// TIA Portal V16 export
// export: Created 2022-03-28T07:44:04.7254911Z, ExportSetting WithDefaults, DisplayName Totally Integrated Automation Portal, DisplayVersion V16 Update 5, DisplayName TIA Portal Version Control Interface, DisplayVersion V16 Update 2, DisplayName TIA Portal Openness, DisplayVersion V16 Update 5, DisplayName STEP 7 Professional, DisplayVersion V16 Update 5, DisplayName STEP 7 Safety, DisplayVersion V16, DisplayName WinCC Professional, DisplayVersion V16 Update 5
FUNCTION "fc_02_Outputs" : Void   // FC2, LAD
{ S7_Optimized_Access := 'TRUE' }
VERSION : 0.1
// stored: AutoNumber false, IsIECCheckEnabled false, SetENOAutomatically false, UDAEnableTagReadback false
   VAR_TEMP
      bIsInverted : Bool;
   END_VAR
   VAR_TEMP   // added for the SCL form of the ladder/FBD networks
      _w1 : Bool;
      _w2 : Bool;
      _w3 : Bool;
      _w4 : Bool;
   END_VAR
BEGIN

REGION Network 1: Rele rearme
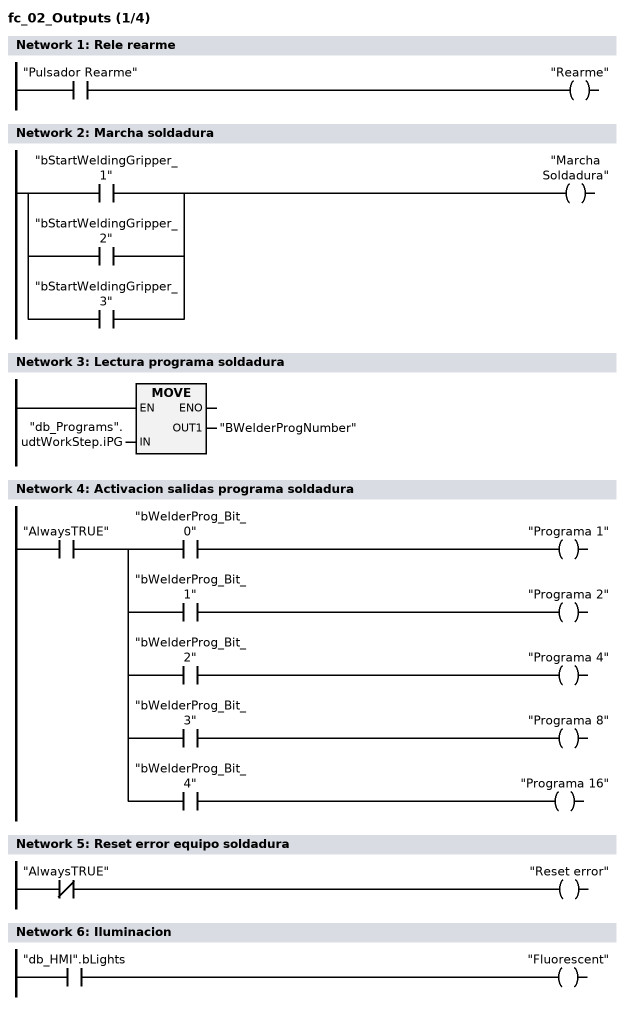
   RUNG wire#powerrail
      Contact( "Pulsador Rearme" )
      Coil( "Rearme" )
   END_RUNG
   // the same network as SCL:
   "Rearme" := "Pulsador Rearme";
END_REGION

REGION Network 2: Marcha soldadura
   RUNG wire#powerrail
      Contact( "bStartWeldingGripper_1" )
      wire#w1
      Coil( "Marcha Soldadura" )
   END_RUNG
   RUNG wire#powerrail
      Contact( "bStartWeldingGripper_2" )
   END_RUNG wire#w1
   RUNG wire#powerrail
      Contact( "bStartWeldingGripper_3" )
   END_RUNG wire#w1
   // the same network as SCL:
   "Marcha Soldadura" := "bStartWeldingGripper_1" OR "bStartWeldingGripper_2" OR "bStartWeldingGripper_3";
END_REGION

REGION Network 3: Lectura programa soldadura
   RUNG wire#powerrail
      Move(in := "db_Programs".udtWorkStep.iPG, out1 => "BWelderProgNumber")
   END_RUNG
   // the same network as SCL:
   "BWelderProgNumber" := "db_Programs".udtWorkStep.iPG;
END_REGION

REGION Network 4: Activacion salidas programa soldadura
   RUNG wire#powerrail
      Contact( "AlwaysTRUE" )
      wire#w1
      Contact( "bWelderProg_Bit_0" )
      Coil( "Programa 1" )
   END_RUNG
   RUNG wire#w1
      Contact( "bWelderProg_Bit_1" )
      Coil( "Programa 2" )
   END_RUNG
   RUNG wire#w1
      Contact( "bWelderProg_Bit_2" )
      Coil( "Programa 4" )
   END_RUNG
   RUNG wire#w1
      Contact( "bWelderProg_Bit_3" )
      Coil( "Programa 8" )
   END_RUNG
   RUNG wire#w1
      Contact( "bWelderProg_Bit_4" )
      Coil( "Programa 16" )
   END_RUNG
   // the same network as SCL:
   "Programa 1" := "AlwaysTRUE" AND "bWelderProg_Bit_0";
   "Programa 2" := "AlwaysTRUE" AND "bWelderProg_Bit_1";
   "Programa 4" := "AlwaysTRUE" AND "bWelderProg_Bit_2";
   "Programa 8" := "AlwaysTRUE" AND "bWelderProg_Bit_3";
   "Programa 16" := "AlwaysTRUE" AND "bWelderProg_Bit_4";
END_REGION

REGION Network 5: Reset error equipo soldadura
   RUNG wire#powerrail
      I_Contact( "AlwaysTRUE" )
      Coil( "Reset error" )
   END_RUNG
   // the same network as SCL:
   "Reset error" := NOT "AlwaysTRUE";
END_REGION

REGION Network 6: Iluminacion
   RUNG wire#powerrail
      Contact( "db_HMI".bLights )
      Coil( "Fluorescent" )
   END_RUNG
   // the same network as SCL:
   "Fluorescent" := "db_HMI".bLights;
END_REGION

REGION Network 7: Pilotos 1
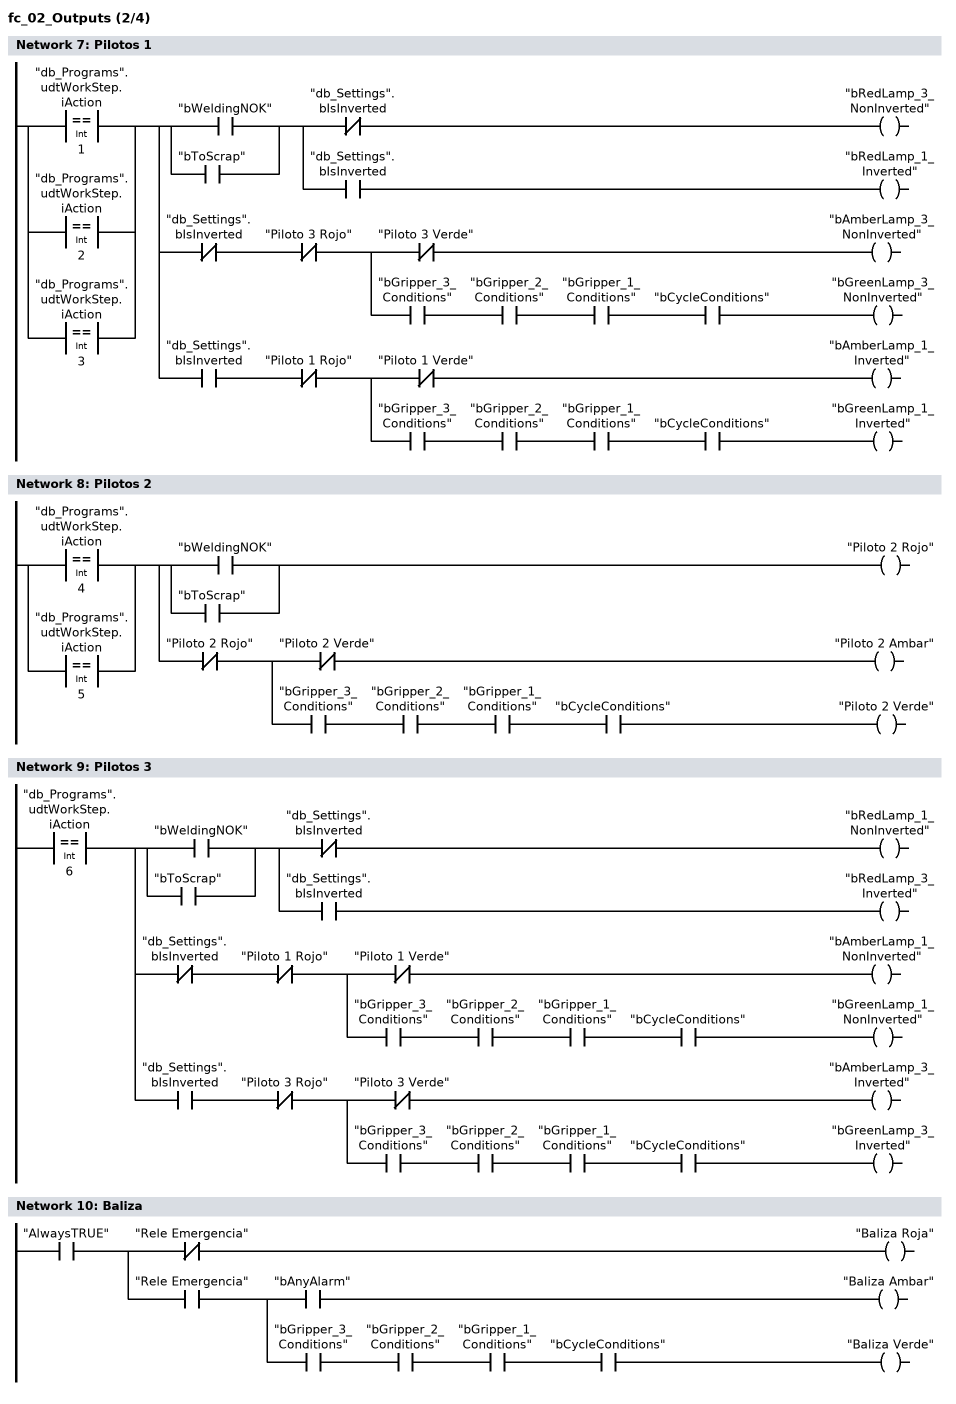
   RUNG wire#powerrail
      { S7_Templates := "SrcType := Int" } EQ_Contact(in1 := "db_Programs".udtWorkStep.iAction, in2 := 1)
      wire#w1
      Contact( "bWeldingNOK" )
      wire#w2
      I_Contact( "db_Settings".bIsInverted )
      Coil( "bRedLamp_3_NonInverted" )
   END_RUNG
   RUNG wire#powerrail
      { S7_Templates := "SrcType := Int" } EQ_Contact(in1 := "db_Programs".udtWorkStep.iAction, in2 := 2)
   END_RUNG wire#w1
   RUNG wire#powerrail
      { S7_Templates := "SrcType := Int" } EQ_Contact(in1 := "db_Programs".udtWorkStep.iAction, in2 := 3)
   END_RUNG wire#w1
   RUNG wire#w1
      Contact( "bToScrap" )
   END_RUNG wire#w2
   RUNG wire#w2
      Contact( "db_Settings".bIsInverted )
      Coil( "bRedLamp_1_Inverted" )
   END_RUNG
   RUNG wire#w1
      I_Contact( "db_Settings".bIsInverted )
      I_Contact( "Piloto 3 Rojo" )
      wire#w3
      I_Contact( "Piloto 3 Verde" )
      Coil( "bAmberLamp_3_NonInverted" )
   END_RUNG
   RUNG wire#w3
      Contact( "bGripper_3_Conditions" )
      Contact( "bGripper_2_Conditions" )
      Contact( "bGripper_1_Conditions" )
      Contact( "bCycleConditions" )
      Coil( "bGreenLamp_3_NonInverted" )
   END_RUNG
   RUNG wire#w1
      Contact( "db_Settings".bIsInverted )
      I_Contact( "Piloto 1 Rojo" )
      wire#w4
      I_Contact( "Piloto 1 Verde" )
      Coil( "bAmberLamp_1_Inverted" )
   END_RUNG
   RUNG wire#w4
      Contact( "bGripper_3_Conditions" )
      Contact( "bGripper_2_Conditions" )
      Contact( "bGripper_1_Conditions" )
      Contact( "bCycleConditions" )
      Coil( "bGreenLamp_1_Inverted" )
   END_RUNG
   // the same network as SCL:
   #_w1 := ("db_Programs".udtWorkStep.iAction = 1) OR ("db_Programs".udtWorkStep.iAction = 2) OR ("db_Programs".udtWorkStep.iAction = 3);
   #_w2 := #_w1 AND ("bWeldingNOK" OR "bToScrap");
   "bRedLamp_3_NonInverted" := #_w2 AND NOT "db_Settings".bIsInverted;
   "bRedLamp_1_Inverted" := #_w2 AND "db_Settings".bIsInverted;
   #_w3 := #_w1 AND NOT "db_Settings".bIsInverted AND NOT "Piloto 3 Rojo";
   "bAmberLamp_3_NonInverted" := #_w3 AND NOT "Piloto 3 Verde";
   "bGreenLamp_3_NonInverted" := #_w3 AND "bGripper_3_Conditions" AND "bGripper_2_Conditions" AND "bGripper_1_Conditions" AND "bCycleConditions";
   #_w4 := #_w1 AND "db_Settings".bIsInverted AND NOT "Piloto 1 Rojo";
   "bAmberLamp_1_Inverted" := #_w4 AND NOT "Piloto 1 Verde";
   "bGreenLamp_1_Inverted" := #_w4 AND "bGripper_3_Conditions" AND "bGripper_2_Conditions" AND "bGripper_1_Conditions" AND "bCycleConditions";
END_REGION

REGION Network 8: Pilotos 2
   RUNG wire#powerrail
      { S7_Templates := "SrcType := Int" } EQ_Contact(in1 := "db_Programs".udtWorkStep.iAction, in2 := 4)
      wire#w1
      Contact( "bWeldingNOK" )
      wire#w2
      Coil( "Piloto 2 Rojo" )
   END_RUNG
   RUNG wire#powerrail
      { S7_Templates := "SrcType := Int" } EQ_Contact(in1 := "db_Programs".udtWorkStep.iAction, in2 := 5)
   END_RUNG wire#w1
   RUNG wire#w1
      Contact( "bToScrap" )
   END_RUNG wire#w2
   RUNG wire#w1
      I_Contact( "Piloto 2 Rojo" )
      wire#w3
      I_Contact( "Piloto 2 Verde" )
      Coil( "Piloto 2 Ambar" )
   END_RUNG
   RUNG wire#w3
      Contact( "bGripper_3_Conditions" )
      Contact( "bGripper_2_Conditions" )
      Contact( "bGripper_1_Conditions" )
      Contact( "bCycleConditions" )
      Coil( "Piloto 2 Verde" )
   END_RUNG
   // the same network as SCL:
   #_w1 := ("db_Programs".udtWorkStep.iAction = 4) OR ("db_Programs".udtWorkStep.iAction = 5);
   "Piloto 2 Rojo" := #_w1 AND ("bWeldingNOK" OR "bToScrap");
   #_w2 := #_w1 AND NOT "Piloto 2 Rojo";
   "Piloto 2 Ambar" := #_w2 AND NOT "Piloto 2 Verde";
   "Piloto 2 Verde" := #_w2 AND "bGripper_3_Conditions" AND "bGripper_2_Conditions" AND "bGripper_1_Conditions" AND "bCycleConditions";
END_REGION

REGION Network 9: Pilotos 3
   RUNG wire#powerrail
      { S7_Templates := "SrcType := Int" } EQ_Contact(in1 := "db_Programs".udtWorkStep.iAction, in2 := 6)
      wire#w1
      Contact( "bWeldingNOK" )
      wire#w2
      I_Contact( "db_Settings".bIsInverted )
      Coil( "bRedLamp_1_NonInverted" )
   END_RUNG
   RUNG wire#w1
      Contact( "bToScrap" )
   END_RUNG wire#w2
   RUNG wire#w2
      Contact( "db_Settings".bIsInverted )
      Coil( "bRedLamp_3_Inverted" )
   END_RUNG
   RUNG wire#w1
      I_Contact( "db_Settings".bIsInverted )
      I_Contact( "Piloto 1 Rojo" )
      wire#w3
      I_Contact( "Piloto 1 Verde" )
      Coil( "bAmberLamp_1_NonInverted" )
   END_RUNG
   RUNG wire#w3
      Contact( "bGripper_3_Conditions" )
      Contact( "bGripper_2_Conditions" )
      Contact( "bGripper_1_Conditions" )
      Contact( "bCycleConditions" )
      Coil( "bGreenLamp_1_NonInverted" )
   END_RUNG
   RUNG wire#w1
      Contact( "db_Settings".bIsInverted )
      I_Contact( "Piloto 3 Rojo" )
      wire#w4
      I_Contact( "Piloto 3 Verde" )
      Coil( "bAmberLamp_3_Inverted" )
   END_RUNG
   RUNG wire#w4
      Contact( "bGripper_3_Conditions" )
      Contact( "bGripper_2_Conditions" )
      Contact( "bGripper_1_Conditions" )
      Contact( "bCycleConditions" )
      Coil( "bGreenLamp_3_Inverted" )
   END_RUNG
   // the same network as SCL:
   #_w1 := "db_Programs".udtWorkStep.iAction = 6;
   #_w2 := #_w1 AND ("bWeldingNOK" OR "bToScrap");
   "bRedLamp_1_NonInverted" := #_w2 AND NOT "db_Settings".bIsInverted;
   "bRedLamp_3_Inverted" := #_w2 AND "db_Settings".bIsInverted;
   #_w3 := #_w1 AND NOT "db_Settings".bIsInverted AND NOT "Piloto 1 Rojo";
   "bAmberLamp_1_NonInverted" := #_w3 AND NOT "Piloto 1 Verde";
   "bGreenLamp_1_NonInverted" := #_w3 AND "bGripper_3_Conditions" AND "bGripper_2_Conditions" AND "bGripper_1_Conditions" AND "bCycleConditions";
   #_w4 := #_w1 AND "db_Settings".bIsInverted AND NOT "Piloto 3 Rojo";
   "bAmberLamp_3_Inverted" := #_w4 AND NOT "Piloto 3 Verde";
   "bGreenLamp_3_Inverted" := #_w4 AND "bGripper_3_Conditions" AND "bGripper_2_Conditions" AND "bGripper_1_Conditions" AND "bCycleConditions";
END_REGION

REGION Network 10: Baliza
   RUNG wire#powerrail
      Contact( "AlwaysTRUE" )
      wire#w1
      I_Contact( "Rele Emergencia" )
      Coil( "Baliza Roja" )
   END_RUNG
   RUNG wire#w1
      Contact( "Rele Emergencia" )
      wire#w2
      Contact( "bAnyAlarm" )
      Coil( "Baliza Ambar" )
   END_RUNG
   RUNG wire#w2
      Contact( "bGripper_3_Conditions" )
      Contact( "bGripper_2_Conditions" )
      Contact( "bGripper_1_Conditions" )
      Contact( "bCycleConditions" )
      Coil( "Baliza Verde" )
   END_RUNG
   // the same network as SCL:
   "Baliza Roja" := "AlwaysTRUE" AND NOT "Rele Emergencia";
   #_w1 := "AlwaysTRUE" AND "Rele Emergencia";
   "Baliza Ambar" := #_w1 AND "bAnyAlarm";
   "Baliza Verde" := #_w1 AND "bGripper_3_Conditions" AND "bGripper_2_Conditions" AND "bGripper_1_Conditions" AND "bCycleConditions";
END_REGION

REGION Network 11: Piloto rearme
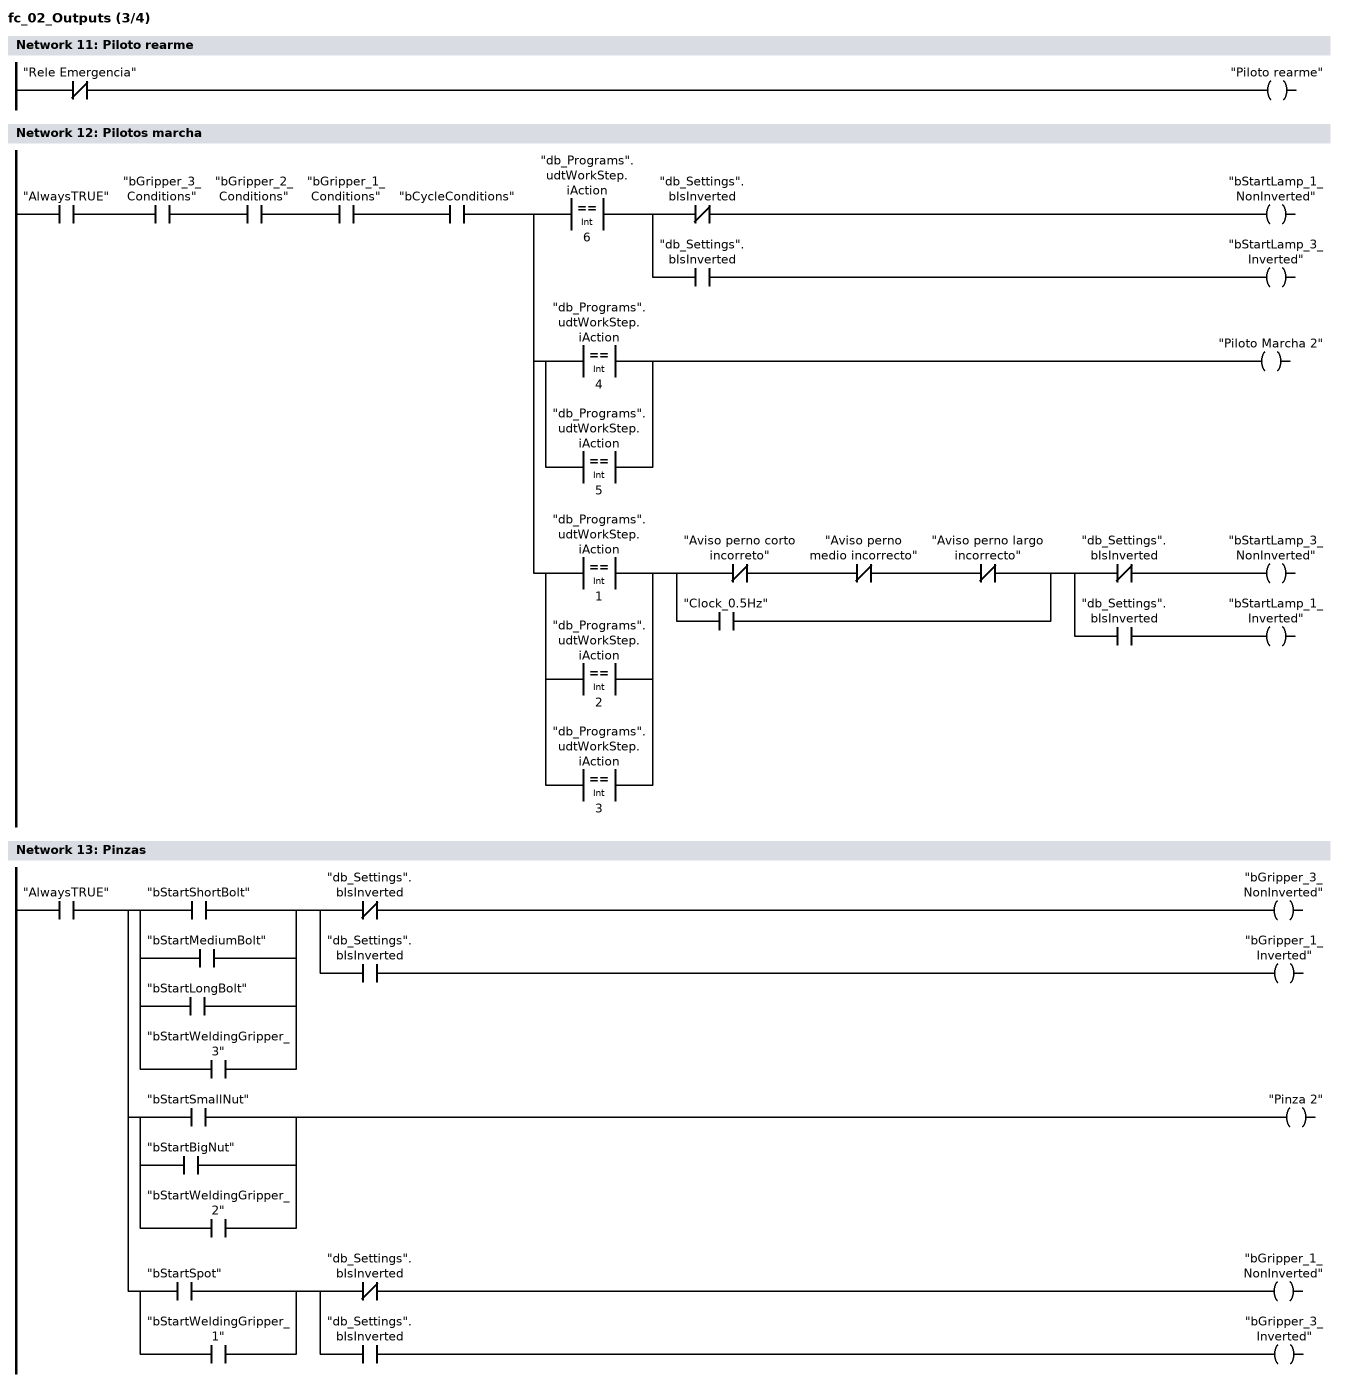
   RUNG wire#powerrail
      I_Contact( "Rele Emergencia" )
      Coil( "Piloto rearme" )
   END_RUNG
   // the same network as SCL:
   "Piloto rearme" := NOT "Rele Emergencia";
END_REGION

REGION Network 12: Pilotos marcha
   RUNG wire#powerrail
      Contact( "AlwaysTRUE" )
      Contact( "bGripper_3_Conditions" )
      Contact( "bGripper_2_Conditions" )
      Contact( "bGripper_1_Conditions" )
      Contact( "bCycleConditions" )
      wire#w1
      { S7_Templates := "SrcType := Int" } EQ_Contact(in1 := "db_Programs".udtWorkStep.iAction, in2 := 6)
      wire#w2
      I_Contact( "db_Settings".bIsInverted )
      Coil( "bStartLamp_1_NonInverted" )
   END_RUNG
   RUNG wire#w2
      Contact( "db_Settings".bIsInverted )
      Coil( "bStartLamp_3_Inverted" )
   END_RUNG
   RUNG wire#w1
      { S7_Templates := "SrcType := Int" } EQ_Contact(in1 := "db_Programs".udtWorkStep.iAction, in2 := 4)
      wire#w3
      Coil( "Piloto Marcha 2" )
   END_RUNG
   RUNG wire#w1
      { S7_Templates := "SrcType := Int" } EQ_Contact(in1 := "db_Programs".udtWorkStep.iAction, in2 := 5)
   END_RUNG wire#w3
   RUNG wire#w1
      { S7_Templates := "SrcType := Int" } EQ_Contact(in1 := "db_Programs".udtWorkStep.iAction, in2 := 1)
      wire#w4
      I_Contact( "Aviso perno corto incorreto" )
      I_Contact( "Aviso perno medio incorrecto" )
      I_Contact( "Aviso perno largo incorrecto" )
      wire#w5
      I_Contact( "db_Settings".bIsInverted )
      Coil( "bStartLamp_3_NonInverted" )
   END_RUNG
   RUNG wire#w1
      { S7_Templates := "SrcType := Int" } EQ_Contact(in1 := "db_Programs".udtWorkStep.iAction, in2 := 2)
   END_RUNG wire#w4
   RUNG wire#w1
      { S7_Templates := "SrcType := Int" } EQ_Contact(in1 := "db_Programs".udtWorkStep.iAction, in2 := 3)
   END_RUNG wire#w4
   RUNG wire#w4
      Contact( "Clock_0.5Hz" )
   END_RUNG wire#w5
   RUNG wire#w5
      Contact( "db_Settings".bIsInverted )
      Coil( "bStartLamp_1_Inverted" )
   END_RUNG
   // the same network as SCL:
   #_w1 := "AlwaysTRUE" AND "bGripper_3_Conditions" AND "bGripper_2_Conditions" AND "bGripper_1_Conditions" AND "bCycleConditions";
   #_w2 := #_w1 AND ("db_Programs".udtWorkStep.iAction = 6);
   "bStartLamp_1_NonInverted" := #_w2 AND NOT "db_Settings".bIsInverted;
   "bStartLamp_3_Inverted" := #_w2 AND "db_Settings".bIsInverted;
   "Piloto Marcha 2" := #_w1 AND (("db_Programs".udtWorkStep.iAction = 4) OR ("db_Programs".udtWorkStep.iAction = 5));
   #_w3 := #_w1 AND (("db_Programs".udtWorkStep.iAction = 1) OR ("db_Programs".udtWorkStep.iAction = 2) OR ("db_Programs".udtWorkStep.iAction = 3)) AND ((NOT "Aviso perno corto incorreto" AND NOT "Aviso perno medio incorrecto" AND NOT "Aviso perno largo incorrecto") OR "Clock_0.5Hz");
   "bStartLamp_3_NonInverted" := #_w3 AND NOT "db_Settings".bIsInverted;
   "bStartLamp_1_Inverted" := #_w3 AND "db_Settings".bIsInverted;
END_REGION

REGION Network 13: Pinzas
   RUNG wire#powerrail
      Contact( "AlwaysTRUE" )
      wire#w1
      Contact( "bStartShortBolt" )
      wire#w2
      I_Contact( "db_Settings".bIsInverted )
      Coil( "bGripper_3_NonInverted" )
   END_RUNG
   RUNG wire#w1
      Contact( "bStartMediumBolt" )
   END_RUNG wire#w2
   RUNG wire#w1
      Contact( "bStartLongBolt" )
   END_RUNG wire#w2
   RUNG wire#w1
      Contact( "bStartWeldingGripper_3" )
   END_RUNG wire#w2
   RUNG wire#w2
      Contact( "db_Settings".bIsInverted )
      Coil( "bGripper_1_Inverted" )
   END_RUNG
   RUNG wire#w1
      Contact( "bStartSmallNut" )
      wire#w3
      Coil( "Pinza 2" )
   END_RUNG
   RUNG wire#w1
      Contact( "bStartBigNut" )
   END_RUNG wire#w3
   RUNG wire#w1
      Contact( "bStartWeldingGripper_2" )
   END_RUNG wire#w3
   RUNG wire#w1
      Contact( "bStartSpot" )
      wire#w4
      I_Contact( "db_Settings".bIsInverted )
      Coil( "bGripper_1_NonInverted" )
   END_RUNG
   RUNG wire#w1
      Contact( "bStartWeldingGripper_1" )
   END_RUNG wire#w4
   RUNG wire#w4
      Contact( "db_Settings".bIsInverted )
      Coil( "bGripper_3_Inverted" )
   END_RUNG
   // the same network as SCL:
   #_w1 := "AlwaysTRUE" AND ("bStartShortBolt" OR "bStartMediumBolt" OR "bStartLongBolt" OR "bStartWeldingGripper_3");
   "bGripper_3_NonInverted" := #_w1 AND NOT "db_Settings".bIsInverted;
   "bGripper_1_Inverted" := #_w1 AND "db_Settings".bIsInverted;
   "Pinza 2" := "AlwaysTRUE" AND ("bStartSmallNut" OR "bStartBigNut" OR "bStartWeldingGripper_2");
   #_w2 := "AlwaysTRUE" AND ("bStartSpot" OR "bStartWeldingGripper_1");
   "bGripper_1_NonInverted" := #_w2 AND NOT "db_Settings".bIsInverted;
   "bGripper_3_Inverted" := #_w2 AND "db_Settings".bIsInverted;
END_REGION

REGION Network 14: Activación Salidas lámparas
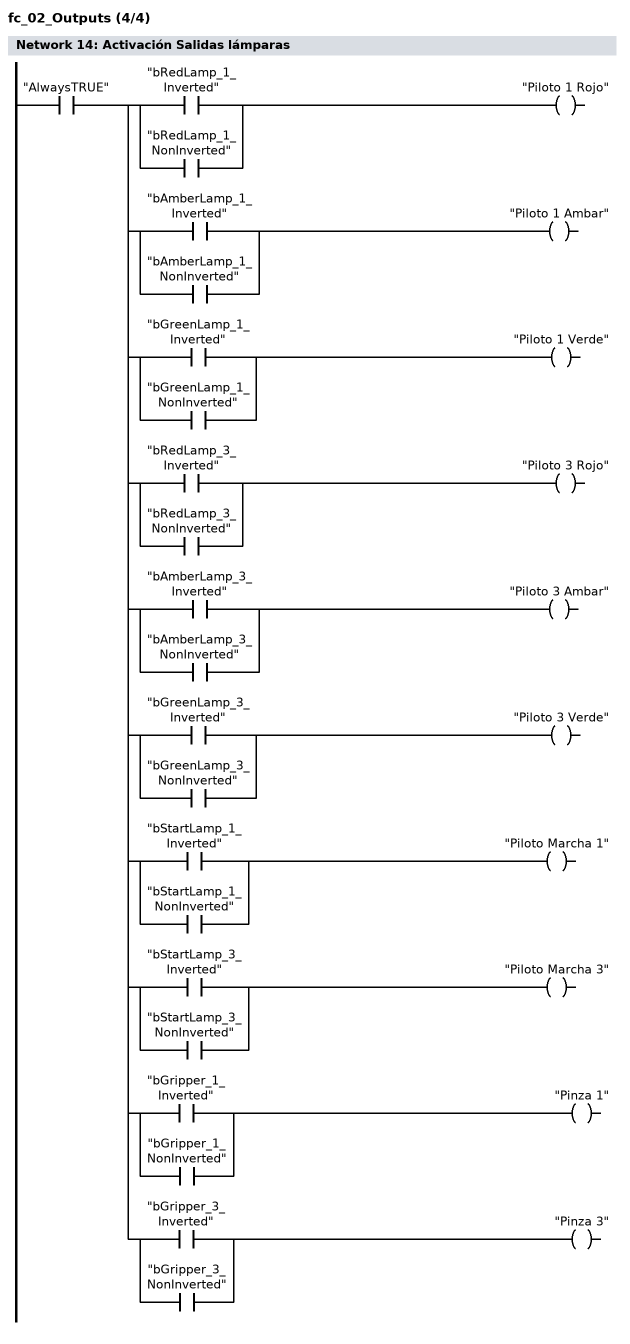
   RUNG wire#powerrail
      Contact( "AlwaysTRUE" )
      wire#w1
      Contact( "bRedLamp_1_Inverted" )
      wire#w2
      Coil( "Piloto 1 Rojo" )
   END_RUNG
   RUNG wire#w1
      Contact( "bRedLamp_1_NonInverted" )
   END_RUNG wire#w2
   RUNG wire#w1
      Contact( "bAmberLamp_1_Inverted" )
      wire#w3
      Coil( "Piloto 1 Ambar" )
   END_RUNG
   RUNG wire#w1
      Contact( "bAmberLamp_1_NonInverted" )
   END_RUNG wire#w3
   RUNG wire#w1
      Contact( "bGreenLamp_1_Inverted" )
      wire#w4
      Coil( "Piloto 1 Verde" )
   END_RUNG
   RUNG wire#w1
      Contact( "bGreenLamp_1_NonInverted" )
   END_RUNG wire#w4
   RUNG wire#w1
      Contact( "bRedLamp_3_Inverted" )
      wire#w5
      Coil( "Piloto 3 Rojo" )
   END_RUNG
   RUNG wire#w1
      Contact( "bRedLamp_3_NonInverted" )
   END_RUNG wire#w5
   RUNG wire#w1
      Contact( "bAmberLamp_3_Inverted" )
      wire#w6
      Coil( "Piloto 3 Ambar" )
   END_RUNG
   RUNG wire#w1
      Contact( "bAmberLamp_3_NonInverted" )
   END_RUNG wire#w6
   RUNG wire#w1
      Contact( "bGreenLamp_3_Inverted" )
      wire#w7
      Coil( "Piloto 3 Verde" )
   END_RUNG
   RUNG wire#w1
      Contact( "bGreenLamp_3_NonInverted" )
   END_RUNG wire#w7
   RUNG wire#w1
      Contact( "bStartLamp_1_Inverted" )
      wire#w8
      Coil( "Piloto Marcha 1" )
   END_RUNG
   RUNG wire#w1
      Contact( "bStartLamp_1_NonInverted" )
   END_RUNG wire#w8
   RUNG wire#w1
      Contact( "bStartLamp_3_Inverted" )
      wire#w9
      Coil( "Piloto Marcha 3" )
   END_RUNG
   RUNG wire#w1
      Contact( "bStartLamp_3_NonInverted" )
   END_RUNG wire#w9
   RUNG wire#w1
      Contact( "bGripper_1_Inverted" )
      wire#w10
      Coil( "Pinza 1" )
   END_RUNG
   RUNG wire#w1
      Contact( "bGripper_1_NonInverted" )
   END_RUNG wire#w10
   RUNG wire#w1
      Contact( "bGripper_3_Inverted" )
      wire#w11
      Coil( "Pinza 3" )
   END_RUNG
   RUNG wire#w1
      Contact( "bGripper_3_NonInverted" )
   END_RUNG wire#w11
   // the same network as SCL:
   "Piloto 1 Rojo" := "AlwaysTRUE" AND ("bRedLamp_1_Inverted" OR "bRedLamp_1_NonInverted");
   "Piloto 1 Ambar" := "AlwaysTRUE" AND ("bAmberLamp_1_Inverted" OR "bAmberLamp_1_NonInverted");
   "Piloto 1 Verde" := "AlwaysTRUE" AND ("bGreenLamp_1_Inverted" OR "bGreenLamp_1_NonInverted");
   "Piloto 3 Rojo" := "AlwaysTRUE" AND ("bRedLamp_3_Inverted" OR "bRedLamp_3_NonInverted");
   "Piloto 3 Ambar" := "AlwaysTRUE" AND ("bAmberLamp_3_Inverted" OR "bAmberLamp_3_NonInverted");
   "Piloto 3 Verde" := "AlwaysTRUE" AND ("bGreenLamp_3_Inverted" OR "bGreenLamp_3_NonInverted");
   "Piloto Marcha 1" := "AlwaysTRUE" AND ("bStartLamp_1_Inverted" OR "bStartLamp_1_NonInverted");
   "Piloto Marcha 3" := "AlwaysTRUE" AND ("bStartLamp_3_Inverted" OR "bStartLamp_3_NonInverted");
   "Pinza 1" := "AlwaysTRUE" AND ("bGripper_1_Inverted" OR "bGripper_1_NonInverted");
   "Pinza 3" := "AlwaysTRUE" AND ("bGripper_3_Inverted" OR "bGripper_3_NonInverted");
END_REGION
END_FUNCTION
